FUNCTION_BLOCK fb_motor_2
VAR_INPUT
	bStart, bStop : BOOL;
	
END_VAR
VAR_OUTPUT
	bStatus : BOOL;
END_VAR
VAR
END_VAR

END_FUNCTION_BLOCK

(* stored: Version 1.1.0.1, ProductVersion 3.1.4024.11
   POU fb_motor_2: Id {23b1ed52-99f0-496b-ac35-592cfa42d18c}, SpecialFunc None *)
